PROGRAM MAIN

ExampleJSON_PRG();

END_PROGRAM

(* stored: Version 1.1.0.1
   POU MAIN: Id {a20f3b3b-f671-464f-8c4c-317e34e9bada}, SpecialFunc None *)
